FUNCTION_BLOCK FB_Homing_CustomPLC EXTENDS FB_Homing_Base
VAR
// =================================================================================
    // IMPORTANT: FOR THIS BLOCK TO WORK, YOU MUST SET THE FOLLOWING IN NC AXIS PARAMETERS:
    // Reference Mode -> 'Application (PLC code)'
    // =================================================================================
    
    fbReadAppReq  : MC_ReadApplicationRequest;
    // fbMcJog       : MC_Jog;
    // fbSetPosition : MC_SetPosition; 
END_VAR

METHOD Abort
VAR_INPUT
END_VAR
SUPER^.Abort();
END_METHOD

METHOD CyclicLogic
CASE nStep OF
    0: // IDLE
    
    10: // READ APPLICATION REQUEST (Placeholder)
        _bBusy := FALSE;
        _bDone := TRUE;
        nStep  := 0;
        
    99: // ERROR HANDLING
        _bBusy    := FALSE;
        _bError   := TRUE;
        _bErrorID := 9999;
        nStep     := 0;
END_CASE
END_METHOD

END_FUNCTION_BLOCK

(* stored: Version 1.1.0.1, ProductVersion 3.1.4024.15
   POU FB_Homing_CustomPLC: Id {67041d96-67cd-4750-9cca-5a2eaf95eb0c}, SpecialFunc None
   Method Abort: Id {12345678-1234-1234-cccc-111111111111}
   Method CyclicLogic: Id {87654321-4321-4321-cccc-222222222222} *)
